TYPE ST_CASE_DefferOuter :
STRUCT
	sID 					: STRING(255);
	ProductionDate 		: STRING(10);
	ProductionTime 		: STRING(8);
	ProductionTimeOffset 	: STRING(6);
	RejectCode 			: STRING(255);
END_STRUCT
END_TYPE

(* stored: Version 1.1.0.1
   DUT ST_CASE_DefferOuter: Id {bf84f0f4-3e39-4aed-968b-e2d5a69d7b01} *)
